KUKA KRL program: Work_2.src, Work_2.dat

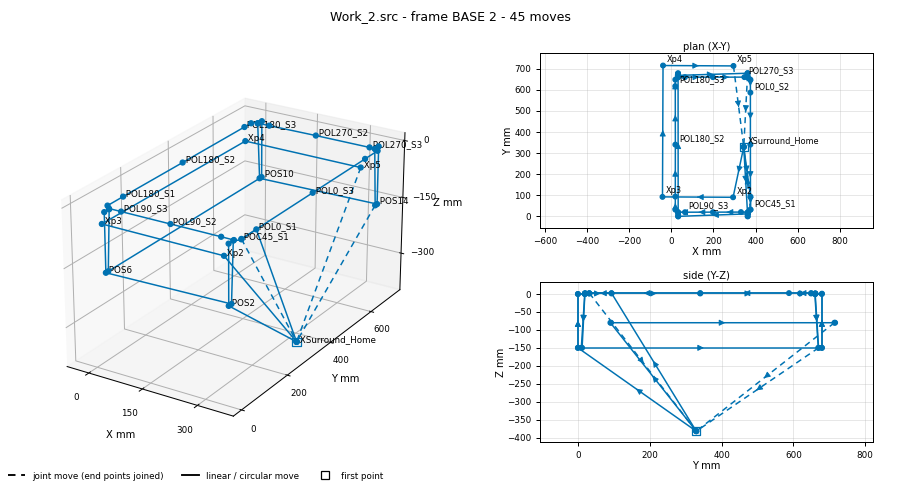
[picture p0: tool path of Work_2.src in frame BASE 2, 45 of 45 moves have a stored position in this frame; points joined in program order, loops and branches not executed]
--- Work_2.src ---
&ACCESS RVO1
&REL 406
&PARAM EDITMASK = *
&PARAM TEMPLATE = C:\KRC\Roboter\Template\vorgabe
&PARAM DISKPATH = KRC:\R1\KRL_HanGao\HG
DEF Work_2( )
;FOLD INI;%{PE}
  ;FOLD BASISTECH INI
    GLOBAL INTERRUPT DECL 3 WHEN $STOPMESS==TRUE DO IR_STOPM ( )
    INTERRUPT ON 3
    BAS (#INITMOV,0 )
  ;ENDFOLD (BASISTECH INI)
  ;FOLD USER INI
    ;Make your modifications here

  ;ENDFOLD (USER INI)
;ENDFOLD (INI)

;FOLD Vision.Vision_Ini ;%{PE}%MKUKATPUSER




EKRL_Vision_Int_Data("Xml_Ini_Data")


;ENDFOLD
;loop
;FOLD PTP Surround_Home Vel=20 % PDAT1 Tool[2]:Work_Tool Base[2]:B_2;%{PE}%R 8.3.48,%MKUKATPBASIS,%CMOVE,%VPTP,%P 1:PTP, 2:Surround_Home, 3:, 5:20, 7:PDAT1
$BWDSTART=FALSE
PDAT_ACT=PPDAT1
FDAT_ACT=FSurround_Home
BAS(#PTP_PARAMS,20)
PTP XSurround_Home
;ENDFOLD


;FOLD Vision.Camera_Offset Camera_NAME :P2, Area:45, Work:2;%{PE}%MKUKATPUSER

 HanGao_Camera_Offset(#Calibration ,1,2,XP2)





;ENDFOLD
;FOLD LIN p2 Vel=0.5 m/s CPDAT1 Tool[2]:Work_Tool Base[2]:Work_2 ;%{PE}
;FOLD Parameters ;%{h}
;Params IlfProvider=kukaroboter.basistech.inlineforms.movement.old; Kuka.IsGlobalPoint=False; Kuka.PointName=p2; Kuka.BlendingEnabled=False; Kuka.MoveDataName=CPDAT1; Kuka.VelocityPath=0.5; Kuka.CurrentCDSetIndex=0; Kuka.MovementParameterFieldEnabled=True; IlfCommand=LIN
;ENDFOLD
$BWDSTART = FALSE
LDAT_ACT = LCPDAT1
FDAT_ACT = Fp2
BAS(#CP_PARAMS, 0.5)
SET_CD_PARAMS (0)
LIN Xp2
;ENDFOLD
;FOLD Vision.Find_Model Work:2, Area:45;%{PE}%MKUKATPUSER



EKRL_Find_Model_Send("Xml_Vision_Model",2,1)



;ENDFOLD


;FOLD Vision.Camera_Offset Camera_NAME :P3, Area:135, Work:2;%{PE}%MKUKATPUSER

 HanGao_Camera_Offset(#Calibration ,2,2,XP3)





;ENDFOLD
;FOLD LIN p3 Vel=0.5 m/s CPDAT2 Tool[2]:Work_Tool Base[2]:Work_2 ;%{PE}
;FOLD Parameters ;%{h}
;Params IlfProvider=kukaroboter.basistech.inlineforms.movement.old; Kuka.IsGlobalPoint=False; Kuka.PointName=p3; Kuka.BlendingEnabled=False; Kuka.MoveDataName=CPDAT2; Kuka.VelocityPath=0.5; Kuka.CurrentCDSetIndex=0; Kuka.MovementParameterFieldEnabled=True; IlfCommand=LIN
;ENDFOLD
$BWDSTART = FALSE
LDAT_ACT = LCPDAT2
FDAT_ACT = Fp3
BAS(#CP_PARAMS, 0.5)
SET_CD_PARAMS (0)
LIN Xp3
;ENDFOLD
;FOLD Vision.Find_Model Work:2, Area:135;%{PE}%MKUKATPUSER



EKRL_Find_Model_Send("Xml_Vision_Model",2,2)



;ENDFOLD


;FOLD Vision.Camera_Offset Camera_NAME :P4, Area:225, Work:2;%{PE}%MKUKATPUSER

 HanGao_Camera_Offset(#Calibration ,3,2,XP4)





;ENDFOLD
;FOLD LIN p4 Vel=0.5 m/s CPDAT3 Tool[2]:Work_Tool Base[2]:Work_2 ;%{PE}
;FOLD Parameters ;%{h}
;Params IlfProvider=kukaroboter.basistech.inlineforms.movement.old; Kuka.IsGlobalPoint=False; Kuka.PointName=p4; Kuka.BlendingEnabled=False; Kuka.MoveDataName=CPDAT3; Kuka.VelocityPath=0.5; Kuka.CurrentCDSetIndex=0; Kuka.MovementParameterFieldEnabled=True; IlfCommand=LIN
;ENDFOLD
$BWDSTART = FALSE
LDAT_ACT = LCPDAT3
FDAT_ACT = Fp4
BAS(#CP_PARAMS, 0.5)
SET_CD_PARAMS (0)
LIN Xp4
;ENDFOLD
;FOLD Vision.Find_Model Work:2, Area:225;%{PE}%MKUKATPUSER



EKRL_Find_Model_Send("Xml_Vision_Model",2,3)



;ENDFOLD


;FOLD Vision.Camera_Offset Camera_NAME :P5, Area:315, Work:2;%{PE}%MKUKATPUSER

 HanGao_Camera_Offset(#Calibration ,4,2,XP5)





;ENDFOLD
;FOLD LIN p5 Vel=0.5 m/s CPDAT4 Tool[2]:Work_Tool Base[2]:Work_2 ;%{PE}
;FOLD Parameters ;%{h}
;Params IlfProvider=kukaroboter.basistech.inlineforms.movement.old; Kuka.IsGlobalPoint=False; Kuka.PointName=p5; Kuka.BlendingEnabled=False; Kuka.MoveDataName=CPDAT4; Kuka.VelocityPath=0.5; Kuka.CurrentCDSetIndex=0; Kuka.MovementParameterFieldEnabled=True; IlfCommand=LIN
;ENDFOLD
$BWDSTART = FALSE
LDAT_ACT = LCPDAT4
FDAT_ACT = Fp5
BAS(#CP_PARAMS, 0.5)
SET_CD_PARAMS (0)
LIN Xp5
;ENDFOLD
;FOLD Vision.Find_Model Work:2, Area:315;%{PE}%MKUKATPUSER



EKRL_Find_Model_Send("Xml_Vision_Model",2,4)



;ENDFOLD
;endloop
;halt
;FOLD PTP Surround_Home Vel=10 % PDAT4 Tool[2]:Work_Tool Base[2]:Work_2 ;%{PE}
;FOLD Parameters ;%{h}
;Params IlfProvider=kukaroboter.basistech.inlineforms.movement.old; Kuka.IsGlobalPoint=False; Kuka.PointName=Surround_Home; Kuka.BlendingEnabled=False; Kuka.MoveDataPtpName=PDAT4; Kuka.VelocityPtp=10; Kuka.CurrentCDSetIndex=0; Kuka.MovementParameterFieldEnabled=True; IlfCommand=PTP
;ENDFOLD
$BWDSTART = FALSE
PDAT_ACT = PPDAT4
FDAT_ACT = FSurround_Home
BAS(#PTP_PARAMS, 10.0)
SET_CD_PARAMS (0)
PTP XSurround_Home
;ENDFOLD
;FOLD Surround_LIN.S_LIN Point: L0_S1, Vel= 0.3 m/s, Point: 90 %, Area: LO, LDAT: L0_L1, OFFSET_NO: 1, Work: N_2 ;%{PE}
; LIN L0_S1POS: X=379.498230, Y=93.8288574, Z=1.00000, A=0.0, B=-20.0000, C=0.0
; LIN Offset POS:X=0.0, Y=0.0, Z=0.0
HanGao_Surr_Calculate( 90, #L0, #L_LIN_POS , POL0_S1, , , L0_Welding_Craft[2,1].Welding_Offset  , , 1, 2 )

HanGao_DAT_ACT(L0_Welding_Craft[2,1],LL0_L1)




FDAT_ACT=FL0_S1
LDAT_ACT=LL0_L1
BAS(#CP_PARAMS,L0_Welding_Craft[2,1].Welding_Speed )
LIN POL0_S1 C_DIS C_DIS
;ENDFOLD
;FOLD Laser_Function.LSON POW= 0 %, Sec= 0 S;%{PE}%MKUKATPUSER



  LSON(0/100,0)


;ENDFOLD
;FOLD Surround_LIN.S_C_LIN Point: C45_S1, Vel= 0.3 m/s, Area: C45, LDAT: C45_L1, Work: N_2 ;%{PE}
; CIR C45_S1POS: X=406.498535, Y=35.6358643, Z=0.0, A=0.0, B=20.0000, C=0.0
; CIR Offset POS:X=0.0, Y=0.0, Z=0.0
HanGao_Surr_Calculate(  , #C45, #C_LIN_POS , POC45_S1, , , C45_Welding_Craft[2,1].Welding_Offset , ,  , 2)

HanGao_DAT_ACT(C45_Welding_Craft[2,1],LC45_L1)




FDAT_ACT=FC45_S1
LDAT_ACT=LC45_L1
BAS(#CP_PARAMS, C45_Welding_Craft[2,1].Welding_Speed )
LIN POC45_S1 C_DIS C_DIS
;ENDFOLD
;FOLD Surround_CIR.S_C_CIR Point:PM3, PE3, Vel=.04m/s, Angle Area: C45, Work: N_2;%{PE}%MKUKATPUSER

; CIR MID POS:PM3 : X=0, Y=0, Z=0, A=0, B=0, C=0
; CIR END POS:PE3 : X=0, Y=0, Z=0, A=0, B=0, C=0
; CIR_MID_OFFSET  : X=0, Y=0, Z=0
; CIR_END_OFFSET  : X=0, Y=0, Z=0
HanGao_Surr_Calculate(  , #C45, #C_CIR_POS ,  , POPM3, POPE3 , C45_Welding_Craft[2,2].Welding_Offset  , C45_Welding_Craft[2, 3].Welding_Offset  ,  , 2)
TRIGGER WHEN PATH=0 DELAY=0 DO $ANOUT[1]=C45_Welding_Craft[2,3].Welding_Power/100

LPM3.VEL=C45_Welding_Craft[2,3].Welding_Speed
LPM3.ACC=C45_Welding_Craft[2,3].Welding_ACC
LPM3.APO_DIST=C45_Welding_Craft[2,3].Welding_CDIS

FDAT_ACT=FPE3
LDAT_ACT=LPM3
BAS(#CP_PARAMS,C45_Welding_Craft[2,3].Welding_Speed )
CIRC POPM3, POPE3 C_DIS C_DIS

;ENDFOLD
;FOLD Surround_LIN.S_LIN Point: L90_S1, Vel= 0.025 m/s, Point: 10 %, Area: L90, LDAT: L90_L1, OFFSET_NO: 1, Work: N_2 ;%{PE}
; LIN L90_S1POS: X=330.358398, Y=17.8462887, Z=1.00000, A=0.0, B=0.0, C=20.0000
; LIN Offset POS:X=0.0, Y=0.200000, Z=0.0
HanGao_Surr_Calculate( 10, #L90, #L_LIN_POS , POL90_S1, , , L90_Welding_Craft[2,1].Welding_Offset  , , 1, 2 )

HanGao_DAT_ACT(L90_Welding_Craft[2,1],LL90_L1)




FDAT_ACT=FL90_S1
LDAT_ACT=LL90_L1
BAS(#CP_PARAMS,L90_Welding_Craft[2,1].Welding_Speed )
LIN POL90_S1 C_DIS C_DIS
;ENDFOLD
;FOLD Surround_LIN.S_LIN Point: L90_S2, Vel= 0.025 m/s, Point: 50 %, Area: L90, LDAT: L90_L2, OFFSET_NO: 2, Work: N_2 ;%{PE}
; LIN L90_S2POS: X=0.0, Y=0.0, Z=0.0, A=0.0, B=0.0, C=0.0
; LIN Offset POS:X=0.0, Y=0.200000, Z=0.0
HanGao_Surr_Calculate( 50, #L90, #L_LIN_POS , POL90_S2, , , L90_Welding_Craft[2,2].Welding_Offset  , , 2, 2 )

HanGao_DAT_ACT(L90_Welding_Craft[2,2],LL90_L2)




FDAT_ACT=FL90_S2
LDAT_ACT=LL90_L2
BAS(#CP_PARAMS,L90_Welding_Craft[2,2].Welding_Speed )
LIN POL90_S2 C_DIS C_DIS
;ENDFOLD
;FOLD Surround_LIN.S_LIN Point: L90_S3, Vel= 0.025 m/s, Point: 90 %, Area: L90, LDAT: L90_L3, OFFSET_NO: 3, Work: N_2 ;%{PE}
; LIN L90_S3POS: X=0.0, Y=0.0, Z=0.0, A=0.0, B=0.0, C=0.0
; LIN Offset POS:X=0.0, Y=0.200000, Z=0.0
HanGao_Surr_Calculate( 90, #L90, #L_LIN_POS , POL90_S3, , , L90_Welding_Craft[2,3].Welding_Offset  , , 3, 2 )

HanGao_DAT_ACT(L90_Welding_Craft[2,3],LL90_L3)




FDAT_ACT=FL90_S3
LDAT_ACT=LL90_L3
BAS(#CP_PARAMS,L90_Welding_Craft[2,3].Welding_Speed )
LIN POL90_S3 C_DIS C_DIS
;ENDFOLD
;FOLD Surround_LIN.S_C_LIN Point: C135_S1, Vel= 0.2 m/s, Area: C135, LDAT: C135_L1, Work: N_2 ;%{PE}
; CIR C135_S1POS: X=0.0, Y=0.0, Z=0.0, A=0.0, B=0.0, C=0.0
; CIR Offset POS:X=-0.500000, Y=0.0, Z=0.0
HanGao_Surr_Calculate(  , #C135, #C_LIN_POS , POC135_S1, , , C135_Welding_Craft[2,1].Welding_Offset , ,  , 2)

HanGao_DAT_ACT(C135_Welding_Craft[2,1],LC135_L1)




FDAT_ACT=FC135_S1
LDAT_ACT=LC135_L1
BAS(#CP_PARAMS, C135_Welding_Craft[2,1].Welding_Speed )
LIN POC135_S1 C_DIS C_DIS
;ENDFOLD
;FOLD Surround_CIR.S_C_CIR Point: PM4, PE4, Vel= 0.012 m/s, Angle Area: C135, Work: N_2 ;%{PE}
; CIR MID POS:PM4 : X=22.6620, Y=25.2540, Z=1.00000, A=0.0, B=0.0, C=0.0
; CIR END POS:PE4 : X=20.6667957, Y=33.6577797, Z=0.0, A=0.0, B=-20.0000, C=0.0
; CIR_MID_OFFSET  : X=0.0, Y=0.0, Z=0.0
; CIR_END_OFFSET  : X=0.500000, Y=0.0, Z=-1.00000
HanGao_Surr_Calculate(  , #C135, #C_CIR_POS ,  , POPM4, POPE4 , C135_Welding_Craft[2,2].Welding_Offset  , C135_Welding_Craft[2, 3].Welding_Offset  ,  , 2)

HanGao_DAT_ACT(C135_Welding_Craft[2,3],LPM4)




FDAT_ACT=FPE4
LDAT_ACT=LPM4
BAS(#CP_PARAMS,C135_Welding_Craft[2,3].Welding_Speed )
CIRC POPM4, POPE4 C_DIS C_DIS
;ENDFOLD
;FOLD Surround_LIN.S_LIN Point: L180_S1, Vel= 0.025 m/s, Point: 10 %, Area: L180, LDAT: L180_L1, OFFSET_NO: 1, Work: N_2 ;%{PE}
; LIN L180_S1POS: X=20.5413361, Y=95.3976288, Z=0.0, A=0.0, B=-20.0000, C=0.0
; LIN Offset POS:X=0.0, Y=0.0, Z=-1.00000
HanGao_Surr_Calculate( 10, #L180, #L_LIN_POS , POL180_S1, , , L180_Welding_Craft[2,1].Welding_Offset  , , 1, 2 )

HanGao_DAT_ACT(L180_Welding_Craft[2,1],LL180_L1)




FDAT_ACT=FL180_S1
LDAT_ACT=LL180_L1
BAS(#CP_PARAMS,L180_Welding_Craft[2,1].Welding_Speed )
LIN POL180_S1 C_DIS C_DIS
;ENDFOLD
;FOLD Surround_LIN.S_LIN Point: L180_S2, Vel= 0.03 m/s, Point: 50 %, Area: L180, LDAT: L180_L2, OFFSET_NO: 2, Work: N_2 ;%{PE}
; LIN L180_S2POS: X=22.3395, Y=342.357025, Z=0.0, A=0.0, B=-20.0000, C=0.0
; LIN Offset POS:X=0.300000, Y=0.0, Z=-1.00000
HanGao_Surr_Calculate( 50, #L180, #L_LIN_POS , POL180_S2, , , L180_Welding_Craft[2,2].Welding_Offset  , , 2, 2 )

HanGao_DAT_ACT(L180_Welding_Craft[2,2],LL180_L2)




FDAT_ACT=FL180_S2
LDAT_ACT=LL180_L2
BAS(#CP_PARAMS,L180_Welding_Craft[2,2].Welding_Speed )
LIN POL180_S2 C_DIS C_DIS
;ENDFOLD
;FOLD Surround_LIN.S_LIN Point: L180_S3, Vel= 0.03 m/s, Point: 95 %, Area: L180, LDAT: L180_L3, OFFSET_NO: 3, Work: N_2 ;%{PE}
; LIN L180_S3POS: X=24.0249329, Y=620.186340, Z=0.0, A=0.0, B=-20.0000, C=0.0
; LIN Offset POS:X=0.300000, Y=0.0, Z=-1.00000
HanGao_Surr_Calculate( 95, #L180, #L_LIN_POS , POL180_S3, , , L180_Welding_Craft[2,3].Welding_Offset  , , 3, 2 )

HanGao_DAT_ACT(L180_Welding_Craft[2,3],LL180_L3)




FDAT_ACT=FL180_S3
LDAT_ACT=LL180_L3
BAS(#CP_PARAMS,L180_Welding_Craft[2,3].Welding_Speed )
LIN POL180_S3 C_DIS C_DIS
;ENDFOLD
;FOLD Surround_LIN.S_C_LIN Point: C225_S1, Vel= 0.2 m/s, Area: C225, LDAT: C225_L1, Work: N_2 ;%{PE}
; CIR C225_S1POS: X=24.2122040, Y=651.056274, Z=0.0, A=0.0, B=-20.0000, C=0.0
; CIR Offset POS:X=-0.500000, Y=0.0, Z=0.0
HanGao_Surr_Calculate(  , #C225, #C_LIN_POS , POC225_S1, , , C225_Welding_Craft[2,1].Welding_Offset , ,  , 2)

HanGao_DAT_ACT(C225_Welding_Craft[2,1],LC225_L1)




FDAT_ACT=FC225_S1
LDAT_ACT=LC225_L1
BAS(#CP_PARAMS, C225_Welding_Craft[2,1].Welding_Speed )
LIN POC225_S1 C_DIS C_DIS
;ENDFOLD
;FOLD Surround_CIR.S_C_CIR Point: PM5, PE5, Vel= 0.012 m/s, Angle Area: C225, Work: N_2 ;%{PE}
; CIR MID POS:PM5 : X=28.3490, Y=660.056, Z=1.00000, A=0.0, B=0.0, C=0.0
; CIR END POS:PE5 : X=35.9848671, Y=663.799744, Z=1.00000, A=0.0, B=0.0, C=-20.0000
; CIR_MID_OFFSET  : X=0.0, Y=0.500000, Z=0.0
; CIR_END_OFFSET  : X=0.0, Y=0.800000, Z=0.0
HanGao_Surr_Calculate(  , #C225, #C_CIR_POS ,  , POPM5, POPE5 , C225_Welding_Craft[2,2].Welding_Offset  , C225_Welding_Craft[2, 3].Welding_Offset  ,  , 2)

HanGao_DAT_ACT(C225_Welding_Craft[2,3],LPM5)




FDAT_ACT=FPE5
LDAT_ACT=LPM5
BAS(#CP_PARAMS,C225_Welding_Craft[2,3].Welding_Speed )
CIRC POPM5, POPE5 C_DIS C_DIS
;ENDFOLD
;FOLD Surround_LIN.S_LIN Point: L270_S1, Vel= 0.025 m/s, Point: 10 %, Area: L270, LDAT: l270_L1, OFFSET_NO: 1, Work: N_2 ;%{PE}
; LIN L270_S1POS: X=69.2440872, Y=662.843689, Z=1.00000, A=0.0, B=0.0, C=-20.0000
; LIN Offset POS:X=0.0, Y=0.0, Z=0.0
HanGao_Surr_Calculate( 10, #L270, #L_LIN_POS , POL270_S1, , , L270_Welding_Craft[2,1].Welding_Offset  , , 1, 2 )

HanGao_DAT_ACT(L270_Welding_Craft[2,1],Ll270_L1)




FDAT_ACT=FL270_S1
LDAT_ACT=Ll270_L1
BAS(#CP_PARAMS,L270_Welding_Craft[2,1].Welding_Speed )
LIN POL270_S1 C_DIS C_DIS
;ENDFOLD
;FOLD Surround_LIN.S_LIN Point: L270_S2, Vel= 0.03 m/s, Point: 50 %, Area: L270, LDAT: L270_L2, OFFSET_NO: 2, Work: N_2 ;%{PE}
; LIN L270_S2POS: X=202.280975, Y=661.419495, Z=1.00000, A=0.0, B=0.0, C=-20.0000
; LIN Offset POS:X=0.0, Y=-0.800000, Z=0.0
HanGao_Surr_Calculate( 50, #L270, #L_LIN_POS , POL270_S2, , , L270_Welding_Craft[2,2].Welding_Offset  , , 2, 2 )

HanGao_DAT_ACT(L270_Welding_Craft[2,2],LL270_L2)




FDAT_ACT=FL270_S2
LDAT_ACT=LL270_L2
BAS(#CP_PARAMS,L270_Welding_Craft[2,2].Welding_Speed )
LIN POL270_S2 C_DIS C_DIS
;ENDFOLD
;FOLD Surround_LIN.S_LIN Point: L270_S3, Vel= 0.03 m/s, Point: 95 %, Area: L270, LDAT: L270_L3, OFFSET_NO: 3, Work: N_2 ;%{PE}
; LIN L270_S3POS: X=351.947479, Y=660.717285, Z=1.00000, A=0.0, B=0.0, C=-20.0000
; LIN Offset POS:X=0.0, Y=-0.800000, Z=0.0
HanGao_Surr_Calculate( 95, #L270, #L_LIN_POS , POL270_S3, , , L270_Welding_Craft[2,3].Welding_Offset  , , 3, 2 )

HanGao_DAT_ACT(L270_Welding_Craft[2,3],LL270_L3)




FDAT_ACT=FL270_S3
LDAT_ACT=LL270_L3
BAS(#CP_PARAMS,L270_Welding_Craft[2,3].Welding_Speed )
LIN POL270_S3 C_DIS C_DIS
;ENDFOLD
;FOLD Surround_LIN.S_C_LIN Point: C315_S1, Vel= 0.2 m/s, Area: C315, LDAT: C315_L1, Work: N_2 ;%{PE}
; CIR C315_S1POS: X=368.577087, Y=660.939270, Z=1.00000, A=0.0, B=0.0, C=-20.0000
; CIR Offset POS:X=-0.500000, Y=0.0, Z=0.0
HanGao_Surr_Calculate(  , #C315, #C_LIN_POS , POC315_S1, , , C315_Welding_Craft[2,1].Welding_Offset , ,  , 2)

HanGao_DAT_ACT(C315_Welding_Craft[2,1],LC315_L1)




FDAT_ACT=FC315_S1
LDAT_ACT=LC315_L1
BAS(#CP_PARAMS, C315_Welding_Craft[2,1].Welding_Speed )
LIN POC315_S1 C_DIS C_DIS
;ENDFOLD
;FOLD Surround_CIR.S_C_CIR Point: PM7, PE7, Vel= 0.012 m/s, Angle Area: C315, Work: N_2 ;%{PE}
; CIR MID POS:PM7 : X=377.618, Y=656.195, Z=1.00000, A=0.0, B=0.0, C=0.0
; CIR END POS:PE7 : X=380.001862, Y=649.383240, Z=1.00000, A=0.0, B=20.0000, C=0.0
; CIR_MID_OFFSET  : X=0.0, Y=-0.500000, Z=0.0
; CIR_END_OFFSET  : X=-0.500000, Y=0.0, Z=0.0
HanGao_Surr_Calculate(  , #C315, #C_CIR_POS ,  , POPM7, POPE7 , C315_Welding_Craft[2,2].Welding_Offset  , C315_Welding_Craft[2, 3].Welding_Offset  ,  , 2)

HanGao_DAT_ACT(C315_Welding_Craft[2,3],LPM7)




FDAT_ACT=FPE7
LDAT_ACT=LPM7
BAS(#CP_PARAMS,C315_Welding_Craft[2,3].Welding_Speed )
CIRC POPM7, POPE7 C_DIS C_DIS
;ENDFOLD
;FOLD Surround_LIN.S_LIN Point: L0_S2, Vel= 0.03 m/s, Point: 10 %, Area: LO, LDAT: L0_L2, OFFSET_NO: 2, Work: N_2 ;%{PE}
; LIN L0_S2POS: X=379.614777, Y=587.556091, Z=1.00000, A=0.0, B=20.0000, C=0.0
; LIN Offset POS:X=-0.500000, Y=0.0, Z=0.0
HanGao_Surr_Calculate( 10, #L0, #L_LIN_POS , POL0_S2, , , L0_Welding_Craft[2,2].Welding_Offset  , , 2, 2 )

HanGao_DAT_ACT(L0_Welding_Craft[2,2],LL0_L2)




FDAT_ACT=FL0_S2
LDAT_ACT=LL0_L2
BAS(#CP_PARAMS,L0_Welding_Craft[2,2].Welding_Speed )
LIN POL0_S2 C_DIS C_DIS
;ENDFOLD
;FOLD Surround_LIN.S_LIN Point: L0_S3, Vel= 0.03 m/s, Point: 50 %, Area: LO, LDAT: L0_L3, OFFSET_NO: 3, Work: N_2 ;%{PE}
; LIN L0_S3POS: X=378.066498, Y=340.247498, Z=1.00000, A=0.0, B=20.0000, C=0.0
; LIN Offset POS:X=-0.500000, Y=0.0, Z=0.0
HanGao_Surr_Calculate( 50, #L0, #L_LIN_POS , POL0_S3, , , L0_Welding_Craft[2,3].Welding_Offset  , , 3, 2 )

HanGao_DAT_ACT(L0_Welding_Craft[2,3],LL0_L3)




FDAT_ACT=FL0_S3
LDAT_ACT=LL0_L3
BAS(#CP_PARAMS,L0_Welding_Craft[2,3].Welding_Speed )
LIN POL0_S3 C_DIS C_DIS
;ENDFOLD
;FOLD Surround_LIN.S_LIN Point: L0_S4, Vel= 0.04 m/s, Point: 100 %, Area: LO, LDAT: L0_L4, OFFSET_NO: 4, Work: N_2 ;%{PE}
; LIN L0_S4POS: X=375.599823, Y=62.1482544, Z=2.50000, A=0.0, B=20.0000, C=0.0
; LIN Offset POS:X=-0.200000, Y=0.0, Z=1.00000
HanGao_Surr_Calculate( 100, #L0, #L_LIN_POS , POL0_S4, , , L0_Welding_Craft[2,4].Welding_Offset  , , 4, 2 )

HanGao_DAT_ACT(L0_Welding_Craft[2,4],LL0_L4)




FDAT_ACT=FL0_S4
LDAT_ACT=LL0_L4
BAS(#CP_PARAMS,L0_Welding_Craft[2,4].Welding_Speed )
LIN POL0_S4 C_DIS C_DIS
;ENDFOLD
;FOLD Laser_Function.LSOFF ;%{PE}%MKUKATPUSER


   LSOFF()


;ENDFOLD


;FOLD PTP Surround_Home Vel=10 % PDAT2 Tool[2]:Work_Tool Base[2]:B_2;%{PE}%R 8.3.48,%MKUKATPBASIS,%CMOVE,%VPTP,%P 1:PTP, 2:Surround_Home, 3:, 5:10, 7:PDAT2
$BWDSTART=FALSE
PDAT_ACT=PPDAT2
FDAT_ACT=FSurround_Home
BAS(#PTP_PARAMS,10)
PTP XSurround_Home
;ENDFOLD
if (false) THEN
;halt
;return
;FOLD Short_Craft.S_LIN Point: S2, Vel= 0.5 m/s, Area: N45, Short_Pos: Safety, Point: 50 %, LDAT: L2, Work: N_2 ;%{PE}
; LIN S2POS: X=363.220, Y=-0.316000, Z=-150.000, A=0.0, B=0.0, C=0.0
; LIN Offset POS:X=0.0, Y=0.0, Z=0.0
HanGao_Surr_Calculate( 50, #N45, #L_LIN_POS , POS2, , , N45_Short_Craft[2,1].Welding_Offset  , , 1, 2, N2_Sink_Data.Sink_Type)

HanGao_DAT_ACT(N45_Short_Craft[2,1],LL2)




FDAT_ACT=FS2
LDAT_ACT=LL2
BAS(#CP_PARAMS,N45_Short_Craft[2,1].Welding_Speed )
LIN POS2 C_DIS C_DIS
;ENDFOLD
;FOLD Short_Craft.S_LIN Point: S3, Vel= 0.5 m/s, Area: N45, Short_Pos: Start, Point: 50 %, LDAT: L3, Work: N_2 ;%{PE}
; LIN S3POS: X=363.220, Y=-0.316000, Z=0.0, A=0.0, B=0.0, C=0.0
; LIN Offset POS:X=0.0, Y=0.0, Z=0.0
HanGao_Surr_Calculate( 50, #N45, #L_LIN_POS , POS3, , , N45_Short_Craft[2,2].Welding_Offset  , , 2, 2, N2_Sink_Data.Sink_Type)

HanGao_DAT_ACT(N45_Short_Craft[2,2],LL3)




FDAT_ACT=FS3
LDAT_ACT=LL3
BAS(#CP_PARAMS,N45_Short_Craft[2,2].Welding_Speed )
LIN POS3 C_DIS C_DIS
;ENDFOLD
;FOLD Laser_Function.LSON POW= .5 %, Sec= 0 S;%{PE}%MKUKATPUSER



  LSON(.5/100,0)


;ENDFOLD
;FOLD Short_Craft.S_LIN Point: S4, Vel= 0.01 m/s, Area: N45, Short_Pos: End, Point: 50 %, LDAT: L4, Work: N_2 ;%{PE}
; LIN S4POS: X=363.395, Y=19.3140, Z=0.0, A=0.0, B=0.0, C=0.0
; LIN Offset POS:X=0.0, Y=0.0, Z=0.0
HanGao_Surr_Calculate( 50, #N45, #L_LIN_POS , POS4, , , N45_Short_Craft[2,3].Welding_Offset  , , 3, 2, N2_Sink_Data.Sink_Type)

HanGao_DAT_ACT(N45_Short_Craft[2,3],LL4)




FDAT_ACT=FS4
LDAT_ACT=LL4
BAS(#CP_PARAMS,N45_Short_Craft[2,3].Welding_Speed )
LIN POS4 C_DIS C_DIS
;ENDFOLD
;FOLD Short_Craft.S_LIN Point: S5, Vel= 0.5 m/s, Area: N45, Short_Pos: BackWelding, Point: 10 %, LDAT: L5, Work: N_2 ;%{PE}
; LIN S5POS: X=363.323059, Y=11.2466183, Z=-150.000, A=0.0, B=0.0, C=0.0
; LIN Offset POS:X=0.0, Y=0.0, Z=0.0
HanGao_Surr_Calculate( 10, #N45, #L_LIN_POS , POS5, , , N45_Short_Craft[2,4].Welding_Offset  , , 4, 2, N2_Sink_Data.Sink_Type)

HanGao_DAT_ACT(N45_Short_Craft[2,4],LL5)




FDAT_ACT=FS5
LDAT_ACT=LL5
BAS(#CP_PARAMS,N45_Short_Craft[2,4].Welding_Speed )
LIN POS5 C_DIS C_DIS
;ENDFOLD
;FOLD Laser_Function.LSOFF ;%{PE}%MKUKATPUSER


   LSOFF()


;ENDFOLD


;FOLD Short_Craft.S_LIN Point: S6, Vel= 0.5 m/s, Area: N135, Short_Pos: Safety, Point: 50 %, LDAT: L6, Work: N_2 ;%{PE}
; LIN S6POS: X=32.5260, Y=-0.971000, Z=-150.000, A=0.0, B=0.0, C=0.0
; LIN Offset POS:X=0.0, Y=0.0, Z=0.0
HanGao_Surr_Calculate( 50, #N135, #L_LIN_POS , POS6, , , N135_Short_Craft[2,1].Welding_Offset  , , 1, 2, N2_Sink_Data.Sink_Type)

HanGao_DAT_ACT(N135_Short_Craft[2,1],LL6)




FDAT_ACT=FS6
LDAT_ACT=LL6
BAS(#CP_PARAMS,N135_Short_Craft[2,1].Welding_Speed )
LIN POS6 C_DIS C_DIS
;ENDFOLD
;FOLD Short_Craft.S_LIN Point: S7, Vel= 0.5 m/s, Area: N135, Short_Pos: Start, Point: 50 %, LDAT: L7, Work: N_2 ;%{PE}
; LIN S7POS: X=32.5260, Y=-0.971000, Z=0.0, A=0.0, B=0.0, C=0.0
; LIN Offset POS:X=0.0, Y=0.0, Z=0.0
HanGao_Surr_Calculate( 50, #N135, #L_LIN_POS , POS7, , , N135_Short_Craft[2,2].Welding_Offset  , , 2, 2, N2_Sink_Data.Sink_Type)

HanGao_DAT_ACT(N135_Short_Craft[2,2],LL7)




FDAT_ACT=FS7
LDAT_ACT=LL7
BAS(#CP_PARAMS,N135_Short_Craft[2,2].Welding_Speed )
LIN POS7 C_DIS C_DIS
;ENDFOLD
;FOLD Laser_Function.LSON POW= 60 %, Sec= 0 S;%{PE}%MKUKATPUSER



  LSON(60/100,0)


;ENDFOLD
;FOLD Short_Craft.S_LIN Point: S8, Vel= 0.01 m/s, Area: N135, Short_Pos: End, Point: 50 %, LDAT: L8, Work: N_2 ;%{PE}
; LIN S8POS: X=32.3940, Y=18.1940, Z=0.0, A=0.0, B=0.0, C=0.0
; LIN Offset POS:X=0.0, Y=0.0, Z=0.0
HanGao_Surr_Calculate( 50, #N135, #L_LIN_POS , POS8, , , N135_Short_Craft[2,3].Welding_Offset  , , 3, 2, N2_Sink_Data.Sink_Type)

HanGao_DAT_ACT(N135_Short_Craft[2,3],LL8)




FDAT_ACT=FS8
LDAT_ACT=LL8
BAS(#CP_PARAMS,N135_Short_Craft[2,3].Welding_Speed )
LIN POS8 C_DIS C_DIS
;ENDFOLD
;FOLD Short_Craft.S_LIN Point: S9, Vel= 0.5 m/s, Area: N135, Short_Pos: BackWelding, Point: 50 %, LDAT: L9, Work: N_2 ;%{PE}
; LIN S9POS: X=32.4600, Y=8.61150074, Z=-150.000, A=0.0, B=0.0, C=0.0
; LIN Offset POS:X=0.0, Y=0.0, Z=0.0
HanGao_Surr_Calculate( 50, #N135, #L_LIN_POS , POS9, , , N135_Short_Craft[2,4].Welding_Offset  , , 4, 2, N2_Sink_Data.Sink_Type)

HanGao_DAT_ACT(N135_Short_Craft[2,4],LL9)




FDAT_ACT=FS9
LDAT_ACT=LL9
BAS(#CP_PARAMS,N135_Short_Craft[2,4].Welding_Speed )
LIN POS9 C_DIS C_DIS
;ENDFOLD
;FOLD Laser_Function.LSOFF ;%{PE}%MKUKATPUSER


   LSOFF()


;ENDFOLD


;FOLD Short_Craft.S_LIN Point: S10, Vel= 0.5 m/s, Area: N225, Short_Pos: Safety, Point: 50 %, LDAT: L10, Work: N_2 ;%{PE}
; LIN S10POS: X=31.6330, Y=679.439, Z=-150.000, A=0.0, B=0.0, C=0.0
; LIN Offset POS:X=0.0, Y=0.0, Z=0.0
HanGao_Surr_Calculate( 50, #N225, #L_LIN_POS , POS10, , , N225_Short_Craft[2,1].Welding_Offset  , , 1, 2, N2_Sink_Data.Sink_Type)

HanGao_DAT_ACT(N225_Short_Craft[2,1],LL10)




FDAT_ACT=FS10
LDAT_ACT=LL10
BAS(#CP_PARAMS,N225_Short_Craft[2,1].Welding_Speed )
LIN POS10 C_DIS C_DIS
;ENDFOLD
;FOLD Short_Craft.S_LIN Point: S11, Vel= 0.5 m/s, Area: N225, Short_Pos: Start, Point: 50 %, LDAT: L11, Work: N_2 ;%{PE}
; LIN S11POS: X=31.6330, Y=679.439, Z=0.0, A=0.0, B=0.0, C=0.0
; LIN Offset POS:X=0.0, Y=0.0, Z=0.0
HanGao_Surr_Calculate( 50, #N225, #L_LIN_POS , POS11, , , N225_Short_Craft[2,2].Welding_Offset  , , 2, 2, N2_Sink_Data.Sink_Type)

HanGao_DAT_ACT(N225_Short_Craft[2,2],LL11)




FDAT_ACT=FS11
LDAT_ACT=LL11
BAS(#CP_PARAMS,N225_Short_Craft[2,2].Welding_Speed )
LIN POS11 C_DIS C_DIS
;ENDFOLD
;FOLD Laser_Function.LSON POW= 60 %, Sec= 0 S;%{PE}%MKUKATPUSER



  LSON(60/100,0)


;ENDFOLD
;FOLD Short_Craft.S_LIN Point: S12, Vel= 0.01 m/s, Area: N225, Short_Pos: End, Point: 50 %, LDAT: L12, Work: N_2 ;%{PE}
; LIN S12POS: X=31.8670, Y=660.025, Z=0.0, A=0.0, B=0.0, C=0.0
; LIN Offset POS:X=0.0, Y=0.0, Z=0.0
HanGao_Surr_Calculate( 50, #N225, #L_LIN_POS , POS12, , , N225_Short_Craft[2,3].Welding_Offset  , , 3, 2, N2_Sink_Data.Sink_Type)

HanGao_DAT_ACT(N225_Short_Craft[2,3],LL12)




FDAT_ACT=FS12
LDAT_ACT=LL12
BAS(#CP_PARAMS,N225_Short_Craft[2,3].Welding_Speed )
LIN POS12 C_DIS C_DIS
;ENDFOLD
;FOLD Short_Craft.S_LIN Point: S13, Vel= 0.5 m/s, Area: N225, Short_Pos: BackWelding, Point: 50 %, LDAT: L13, Work: N_2 ;%{PE}
; LIN S13POS: X=31.7500, Y=669.732056, Z=-150.000, A=0.0, B=0.0, C=0.0
; LIN Offset POS:X=0.0, Y=0.0, Z=0.0
HanGao_Surr_Calculate( 50, #N225, #L_LIN_POS , POS13, , , N225_Short_Craft[2,4].Welding_Offset  , , 4, 2, N2_Sink_Data.Sink_Type)

HanGao_DAT_ACT(N225_Short_Craft[2,4],LL13)




FDAT_ACT=FS13
LDAT_ACT=LL13
BAS(#CP_PARAMS,N225_Short_Craft[2,4].Welding_Speed )
LIN POS13 C_DIS C_DIS
;ENDFOLD
;FOLD Laser_Function.LSOFF ;%{PE}%MKUKATPUSER


   LSOFF()


;ENDFOLD


;FOLD Short_Craft.S_LIN Point: S14, Vel= 0.5 m/s, Area: N315, Short_Pos: Safety, Point: 50 %, LDAT: L14, Work: N_2 ;%{PE}
; LIN S14POS: X=362.986, Y=679.910, Z=-150.000, A=0.0, B=0.0, C=0.0
; LIN Offset POS:X=0.0, Y=0.0, Z=0.0
HanGao_Surr_Calculate( 50, #N315, #L_LIN_POS , POS14, , , N315_Short_Craft[2,1].Welding_Offset  , , 1, 2, N2_Sink_Data.Sink_Type)

HanGao_DAT_ACT(N315_Short_Craft[2,1],LL14)




FDAT_ACT=FS14
LDAT_ACT=LL14
BAS(#CP_PARAMS,N315_Short_Craft[2,1].Welding_Speed )
LIN POS14 C_DIS C_DIS
;ENDFOLD
;FOLD Short_Craft.S_LIN Point: S15, Vel= 0.5 m/s, Area: N315, Short_Pos: Start, Point: 50 %, LDAT: L15, Work: N_2 ;%{PE}
; LIN S15POS: X=362.986, Y=679.910, Z=1.00000, A=0.0, B=0.0, C=0.0
; LIN Offset POS:X=0.0, Y=0.0, Z=1.00000
HanGao_Surr_Calculate( 50, #N315, #L_LIN_POS , POS15, , , N315_Short_Craft[2,2].Welding_Offset  , , 2, 2, N2_Sink_Data.Sink_Type)

HanGao_DAT_ACT(N315_Short_Craft[2,2],LL15)




FDAT_ACT=FS15
LDAT_ACT=LL15
BAS(#CP_PARAMS,N315_Short_Craft[2,2].Welding_Speed )
LIN POS15 C_DIS C_DIS
;ENDFOLD
;FOLD Laser_Function.LSON POW= 60 %, Sec= 0 S;%{PE}%MKUKATPUSER



  LSON(60/100,0)


;ENDFOLD
;FOLD Short_Craft.S_LIN Point: S16, Vel= 0.01 m/s, Area: N315, Short_Pos: End, Point: 50 %, LDAT: L16, Work: N_2 ;%{PE}
; LIN S16POS: X=363.044, Y=660.468, Z=1.00000, A=0.0, B=0.0, C=0.0
; LIN Offset POS:X=0.0, Y=0.0, Z=1.00000
HanGao_Surr_Calculate( 50, #N315, #L_LIN_POS , POS16, , , N315_Short_Craft[2,3].Welding_Offset  , , 3, 2, N2_Sink_Data.Sink_Type)

HanGao_DAT_ACT(N315_Short_Craft[2,3],LL16)




FDAT_ACT=FS16
LDAT_ACT=LL16
BAS(#CP_PARAMS,N315_Short_Craft[2,3].Welding_Speed )
LIN POS16 C_DIS C_DIS
;ENDFOLD
;FOLD Short_Craft.S_LIN Point: S17, Vel= 0.5 m/s, Area: N315, Short_Pos: BackWelding, Point: 50 %, LDAT: L17, Work: N_2 ;%{PE}
; LIN S17POS: X=363.015, Y=670.188965, Z=-150.000, A=0.0, B=0.0, C=0.0
; LIN Offset POS:X=0.0, Y=0.0, Z=0.0
HanGao_Surr_Calculate( 50, #N315, #L_LIN_POS , POS17, , , N315_Short_Craft[2,4].Welding_Offset  , , 4, 2, N2_Sink_Data.Sink_Type)

HanGao_DAT_ACT(N315_Short_Craft[2,4],LL17)




FDAT_ACT=FS17
LDAT_ACT=LL17
BAS(#CP_PARAMS,N315_Short_Craft[2,4].Welding_Speed )
LIN POS17 C_DIS C_DIS
;ENDFOLD
;FOLD Laser_Function.LSOFF ;%{PE}%MKUKATPUSER


   LSOFF()


;ENDFOLD
endif

;FOLD PTP Surround_Home CONT Vel=30 % PDAT3 Tool[2]:Work_Tool Base[2]:B_2;%{PE}%R 8.3.48,%MKUKATPBASIS,%CMOVE,%VPTP,%P 1:PTP, 2:Surround_Home, 3:C_DIS, 5:30, 7:PDAT3
$BWDSTART=FALSE
PDAT_ACT=PPDAT3
FDAT_ACT=FSurround_Home
BAS(#PTP_PARAMS,30)
PTP XSurround_Home C_DIS
;ENDFOLD
END

--- Work_2.dat ---
&ACCESS RVO1
&REL 406
&PARAM EDITMASK = *
&PARAM TEMPLATE = C:\KRC\Roboter\Template\vorgabe
&PARAM DISKPATH = KRC:\R1\KRL_HanGao\HG
DEFDAT  WORK_2
;FOLD EXTERNAL DECLARATIONS;%{PE}%MKUKATPBASIS,%CEXT,%VCOMMON,%P
;FOLD BASISTECH EXT;%{PE}%MKUKATPBASIS,%CEXT,%VEXT,%P
EXT  BAS (BAS_COMMAND  :IN,REAL  :IN )
DECL INT SUCCESS
;ENDFOLD (BASISTECH EXT)
;FOLD USER EXT;%{E}%MKUKATPUSER,%CEXT,%VEXT,%P
;Make your modifications here

;ENDFOLD (USER EXT)
;ENDFOLD (EXTERNAL DECLARATIONS)
DECL BASIS_SUGG_T LAST_BASIS={POINT1[] "P0                      ",POINT2[] "P0                      ",CP_PARAMS[] "CPDAT0                  ",PTP_PARAMS[] "PDAT0                   ",CONT[] "                        ",CP_VEL[] "2.0                     ",PTP_VEL[] "100                     ",SYNC_PARAMS[] "SYNCDAT                 ",SPL_NAME[] "S0                      ",A_PARAMS[] "ADAT0                   "}
DECL E6POS XSURROUND_HOME={X 343.780548,Y 329.155823,Z -382.275,A 0.441927075,B -0.0416149125,C -0.0704164580,S 2,T 10,E1 0.0,E2 0.0,E3 0.0,E4 0.0,E5 0.0,E6 0.0}
DECL FDAT FSurround_Home={TOOL_NO 2,BASE_NO 2,IPO_FRAME #BASE,POINT2[] " "}
DECL PDAT PPDAT1={VEL 100.000,ACC 20.0000,APO_DIST 100.000,GEAR_JERK 50.0000,EXAX_IGN 0}
DECL PDAT PPDAT2={VEL 100.000,ACC 20.0000,APO_DIST 100.000,GEAR_JERK 50.0000,EXAX_IGN 0}
DECL E6POS POS2={X 362.596,Y -0.482000,Z -150.000,A 0.0,B 0.0,C 0.0}
DECL FDAT FS2={TOOL_NO 2,BASE_NO 2,IPO_FRAME #BASE,POINT2[] " ",TQ_STATE FALSE}
DECL LDAT LL2={VEL 0.500000,ACC 100.000,APO_DIST 0.0,APO_FAC 50.0000,AXIS_VEL 100.000,AXIS_ACC 100.000,ORI_TYP #VAR,CIRC_TYP #BASE,JERK_FAC 50.0000,GEAR_JERK 50.0000,EXAX_IGN 0}
DECL E6POS POS3={X 362.596,Y -0.482000,Z 0.0,A 0.0,B 0.0,C 0.0}
DECL FDAT FS3={TOOL_NO 2,BASE_NO 2,IPO_FRAME #BASE,POINT2[] " ",TQ_STATE FALSE}
DECL LDAT LL3={VEL 0.500000,ACC 100.000,APO_DIST 0.0,APO_FAC 50.0000,AXIS_VEL 100.000,AXIS_ACC 100.000,ORI_TYP #VAR,CIRC_TYP #BASE,JERK_FAC 50.0000,GEAR_JERK 50.0000,EXAX_IGN 0}
DECL E6POS POS4={X 362.546,Y 18.7470,Z 0.0,A 0.0,B 0.0,C 0.0}
DECL FDAT FS4={TOOL_NO 2,BASE_NO 2,IPO_FRAME #BASE,POINT2[] " ",TQ_STATE FALSE}
DECL LDAT LL4={VEL 0.01000000,ACC 100.000,APO_DIST 0.0,APO_FAC 50.0000,AXIS_VEL 100.000,AXIS_ACC 100.000,ORI_TYP #VAR,CIRC_TYP #BASE,JERK_FAC 50.0000,GEAR_JERK 50.0000,EXAX_IGN 0}
DECL E6POS POS5={X 362.566040,Y 11.0408678,Z -150.000,A 0.0,B 0.0,C 0.0}
DECL FDAT FS5={TOOL_NO 2,BASE_NO 2,IPO_FRAME #BASE,POINT2[] " ",TQ_STATE FALSE}
DECL LDAT LL5={VEL 0.500000,ACC 100.000,APO_DIST 0.0,APO_FAC 50.0000,AXIS_VEL 100.000,AXIS_ACC 100.000,ORI_TYP #VAR,CIRC_TYP #BASE,JERK_FAC 50.0000,GEAR_JERK 50.0000,EXAX_IGN 0}
DECL E6POS POPM3={X 372.487,Y 23.7200,Z 1.50000,A 0.0,B 0.0,C 0.0}
DECL E6POS POPE3={X 363.888,Y 19.3187675,Z 1.50000,A 0.0,B 0.0,C 20.0000}
DECL FDAT FPE3={TOOL_NO 2,BASE_NO 2,IPO_FRAME #BASE,POINT2[] " ",TQ_STATE FALSE}
DECL LDAT LPM3={VEL 0.0230000,ACC 100.000,APO_DIST 5.00000,APO_FAC 50.0000,AXIS_VEL 100.000,AXIS_ACC 100.000,ORI_TYP #VAR,CIRC_TYP #BASE,JERK_FAC 50.0000,GEAR_JERK 50.0000,EXAX_IGN 0}
DECL E6POS POS6={X 32.1370,Y -0.736000,Z -150.000,A 0.0,B 0.0,C 0.0}
DECL FDAT FS6={TOOL_NO 2,BASE_NO 2,IPO_FRAME #BASE,POINT2[] " ",TQ_STATE FALSE}
DECL LDAT LL6={VEL 0.500000,ACC 100.000,APO_DIST 0.0,APO_FAC 50.0000,AXIS_VEL 100.000,AXIS_ACC 100.000,ORI_TYP #VAR,CIRC_TYP #BASE,JERK_FAC 50.0000,GEAR_JERK 50.0000,EXAX_IGN 0}
DECL E6POS POS7={X 32.1370,Y -0.736000,Z 0.0,A 0.0,B 0.0,C 0.0}
DECL FDAT FS7={TOOL_NO 2,BASE_NO 2,IPO_FRAME #BASE,POINT2[] " ",TQ_STATE FALSE}
DECL LDAT LL7={VEL 0.500000,ACC 100.000,APO_DIST 0.0,APO_FAC 50.0000,AXIS_VEL 100.000,AXIS_ACC 100.000,ORI_TYP #VAR,CIRC_TYP #BASE,JERK_FAC 50.0000,GEAR_JERK 50.0000,EXAX_IGN 0}
DECL E6POS POS8={X 32.1600,Y 18.4470,Z 0.0,A 0.0,B 0.0,C 0.0}
DECL FDAT FS8={TOOL_NO 2,BASE_NO 2,IPO_FRAME #BASE,POINT2[] " ",TQ_STATE FALSE}
DECL LDAT LL8={VEL 0.01000000,ACC 100.000,APO_DIST 0.0,APO_FAC 50.0000,AXIS_VEL 100.000,AXIS_ACC 100.000,ORI_TYP #VAR,CIRC_TYP #BASE,JERK_FAC 50.0000,GEAR_JERK 50.0000,EXAX_IGN 0}
DECL E6POS POS9={X 32.1485,Y 8.85550117,Z -150.000,A 0.0,B 0.0,C 0.0}
DECL FDAT FS9={TOOL_NO 2,BASE_NO 2,IPO_FRAME #BASE,POINT2[] " ",TQ_STATE FALSE}
DECL LDAT LL9={VEL 0.500000,ACC 100.000,APO_DIST 0.0,APO_FAC 50.0000,AXIS_VEL 100.000,AXIS_ACC 100.000,ORI_TYP #VAR,CIRC_TYP #BASE,JERK_FAC 50.0000,GEAR_JERK 50.0000,EXAX_IGN 0}
DECL E6POS POPM4={X 23.1220,Y 21.6800,Z 1.50000,A 0.0,B 0.0,C 0.0}
DECL E6POS POPE4={X 18.7403107,Y 31.1279984,Z 1.50000,A 0.0,B -20.0000,C 0.0}
DECL FDAT FPE4={TOOL_NO 2,BASE_NO 2,IPO_FRAME #BASE,POINT2[] " ",TQ_STATE FALSE}
DECL LDAT LPM4={VEL 0.0120000,ACC 100.000,APO_DIST 5.00000,APO_FAC 50.0000,AXIS_VEL 100.000,AXIS_ACC 100.000,ORI_TYP #VAR,CIRC_TYP #BASE,JERK_FAC 50.0000,GEAR_JERK 50.0000,EXAX_IGN 0}
DECL E6POS POPM5={X 22.5580,Y 657.793,Z 1.50000,A 0.0,B 0.0,C 0.0}
DECL E6POS POPE5={X 30.8369904,Y 660.939636,Z 0.500000,A 0.0,B 0.0,C -20.0000}
DECL FDAT FPE5={TOOL_NO 2,BASE_NO 2,IPO_FRAME #BASE,POINT2[] " ",TQ_STATE FALSE}
DECL LDAT LPM5={VEL 0.0120000,ACC 100.000,APO_DIST 5.00000,APO_FAC 50.0000,AXIS_VEL 100.000,AXIS_ACC 100.000,ORI_TYP #VAR,CIRC_TYP #BASE,JERK_FAC 50.0000,GEAR_JERK 50.0000,EXAX_IGN 0}
DECL E6POS POPM7={X 370.952026,Y 658.128,Z 2.50000,A 0.0,B 0.0,C 0.0}
DECL E6POS POPE7={X 375.437683,Y 649.261047,Z 2.50000,A 0.0,B 20.0000,C 0.0}
DECL FDAT FPE7={TOOL_NO 2,BASE_NO 2,IPO_FRAME #BASE,POINT2[] " ",TQ_STATE FALSE}
DECL LDAT LPM7={VEL 0.0120000,ACC 100.000,APO_DIST 5.00000,APO_FAC 50.0000,AXIS_VEL 100.000,AXIS_ACC 100.000,ORI_TYP #VAR,CIRC_TYP #BASE,JERK_FAC 50.0000,GEAR_JERK 50.0000,EXAX_IGN 0}
DECL E6POS POS10={X 31.6630,Y 678.803,Z -150.000,A 0.0,B 0.0,C 0.0}
DECL FDAT FS10={TOOL_NO 2,BASE_NO 2,IPO_FRAME #BASE,POINT2[] " ",TQ_STATE FALSE}
DECL LDAT LL10={VEL 0.500000,ACC 100.000,APO_DIST 0.0,APO_FAC 50.0000,AXIS_VEL 100.000,AXIS_ACC 100.000,ORI_TYP #VAR,CIRC_TYP #BASE,JERK_FAC 50.0000,GEAR_JERK 50.0000,EXAX_IGN 0}
DECL E6POS POS11={X 31.6630,Y 678.803,Z 0.0,A 0.0,B 0.0,C 0.0}
DECL FDAT FS11={TOOL_NO 2,BASE_NO 2,IPO_FRAME #BASE,POINT2[] " ",TQ_STATE FALSE}
DECL LDAT LL11={VEL 0.500000,ACC 100.000,APO_DIST 0.0,APO_FAC 50.0000,AXIS_VEL 100.000,AXIS_ACC 100.000,ORI_TYP #VAR,CIRC_TYP #BASE,JERK_FAC 50.0000,GEAR_JERK 50.0000,EXAX_IGN 0}
DECL E6POS POS12={X 31.3610,Y 659.596,Z 0.0,A 0.0,B 0.0,C 0.0}
DECL FDAT FS12={TOOL_NO 2,BASE_NO 2,IPO_FRAME #BASE,POINT2[] " ",TQ_STATE FALSE}
DECL LDAT LL12={VEL 0.01000000,ACC 100.000,APO_DIST 0.0,APO_FAC 50.0000,AXIS_VEL 100.000,AXIS_ACC 100.000,ORI_TYP #VAR,CIRC_TYP #BASE,JERK_FAC 50.0000,GEAR_JERK 50.0000,EXAX_IGN 0}
DECL E6POS POS13={X 31.5120010,Y 669.199463,Z -150.000,A 0.0,B 0.0,C 0.0}
DECL FDAT FS13={TOOL_NO 2,BASE_NO 2,IPO_FRAME #BASE,POINT2[] " ",TQ_STATE FALSE}
DECL LDAT LL13={VEL 0.500000,ACC 100.000,APO_DIST 0.0,APO_FAC 50.0000,AXIS_VEL 100.000,AXIS_ACC 100.000,ORI_TYP #VAR,CIRC_TYP #BASE,JERK_FAC 50.0000,GEAR_JERK 50.0000,EXAX_IGN 0}
DECL E6POS POS14={X 361.885,Y 679.437,Z -150.000,A 0.0,B 0.0,C 0.0}
DECL FDAT FS14={TOOL_NO 2,BASE_NO 2,IPO_FRAME #BASE,POINT2[] " ",TQ_STATE FALSE}
DECL LDAT LL14={VEL 0.500000,ACC 100.000,APO_DIST 0.0,APO_FAC 50.0000,AXIS_VEL 100.000,AXIS_ACC 100.000,ORI_TYP #VAR,CIRC_TYP #BASE,JERK_FAC 50.0000,GEAR_JERK 50.0000,EXAX_IGN 0}
DECL E6POS POS15={X 361.885,Y 679.437,Z 1.00000,A 0.0,B 0.0,C 0.0}
DECL FDAT FS15={TOOL_NO 2,BASE_NO 2,IPO_FRAME #BASE,POINT2[] " ",TQ_STATE FALSE}
DECL LDAT LL15={VEL 0.500000,ACC 100.000,APO_DIST 0.0,APO_FAC 50.0000,AXIS_VEL 100.000,AXIS_ACC 100.000,ORI_TYP #VAR,CIRC_TYP #BASE,JERK_FAC 50.0000,GEAR_JERK 50.0000,EXAX_IGN 0}
DECL E6POS POS16={X 361.560,Y 660.457,Z 1.00000,A 0.0,B 0.0,C 0.0}
DECL FDAT FS16={TOOL_NO 2,BASE_NO 2,IPO_FRAME #BASE,POINT2[] " ",TQ_STATE FALSE}
DECL LDAT LL16={VEL 0.01000000,ACC 100.000,APO_DIST 0.0,APO_FAC 50.0000,AXIS_VEL 100.000,AXIS_ACC 100.000,ORI_TYP #VAR,CIRC_TYP #BASE,JERK_FAC 50.0000,GEAR_JERK 50.0000,EXAX_IGN 0}
DECL E6POS POS17={X 361.722504,Y 669.947,Z -150.000,A 0.0,B 0.0,C 0.0}
DECL FDAT FS17={TOOL_NO 2,BASE_NO 2,IPO_FRAME #BASE,POINT2[] " ",TQ_STATE FALSE}
DECL LDAT LL17={VEL 0.500000,ACC 100.000,APO_DIST 0.0,APO_FAC 50.0000,AXIS_VEL 100.000,AXIS_ACC 100.000,ORI_TYP #VAR,CIRC_TYP #BASE,JERK_FAC 50.0000,GEAR_JERK 50.0000,EXAX_IGN 0}
DECL PDAT PPDAT3={VEL 100.000,ACC 20.0000,APO_DIST 100.000,APO_MODE #CDIS,GEAR_JERK 50.0000,EXAX_IGN 0}
DECL FDAT FL0_S2={TOOL_NO 2,BASE_NO 2,IPO_FRAME #BASE,POINT2[] " ",TQ_STATE FALSE}
DECL E6POS POL0_S2={X 375.372040,Y 587.535706,Z 2.50000,A 0.0,B 20.0000,C 0.0}
DECL FDAT FL0={TOOL_NO 2,BASE_NO 11,IPO_FRAME #BASE,POINT2[] " ",TQ_STATE FALSE}
DECL E6POS POL0_s4={X 375.681305,Y 31.1079712,Z 2.50000,A 0.0,B 20.0000,C 0.0}
DECL FDAT FL0_s4={TOOL_NO 2,BASE_NO 2,IPO_FRAME #BASE,POINT2[] " ",TQ_STATE FALSE}
DECL E6POS POC45_S5={X 404.000,Y 36.0000,Z -1.00000,A 0.0,B 20.0000,C 0.0}
DECL FDAT FC45_S5={TOOL_NO 2,BASE_NO 11,IPO_FRAME #BASE,POINT2[] " ",TQ_STATE FALSE}
DECL E6POS POL0_S1={X 375.946960,Y 92.9332886,Z 2.50000,A 0.0,B 20.0000,C 0.0}
DECL FDAT FL0_S1={TOOL_NO 2,BASE_NO 2,IPO_FRAME #BASE,POINT2[] " ",TQ_STATE FALSE}
DECL E6POS POC45_S1={X 375.881317,Y 31.1079712,Z 1.50000,A 0.0,B 20.0000,C 0.0}
DECL FDAT FC45_S1={TOOL_NO 2,BASE_NO 2,IPO_FRAME #BASE,POINT2[] " ",TQ_STATE FALSE}
DECL LDAT LL0_L1={VEL 0.300000,ACC 100.000,APO_DIST 5.00000,APO_FAC 50.0000,AXIS_VEL 100.000,AXIS_ACC 100.000,ORI_TYP #VAR,CIRC_TYP #BASE,JERK_FAC 50.0000,GEAR_JERK 50.0000,EXAX_IGN 0}
DECL LDAT LC45_L1={VEL 0.300000,ACC 100.000,APO_DIST 5.00000,APO_FAC 50.0000,AXIS_VEL 100.000,AXIS_ACC 100.000,ORI_TYP #VAR,CIRC_TYP #BASE,JERK_FAC 50.0000,GEAR_JERK 50.0000,EXAX_IGN 0}
DECL E6POS POL90_S1={X 330.624,Y 19.5486126,Z 1.50000,A 0.0,B 0.0,C 20.0000}
DECL FDAT FL90_S1={TOOL_NO 2,BASE_NO 2,IPO_FRAME #BASE,POINT2[] " ",TQ_STATE FALSE}
DECL LDAT LL90_L1={VEL 0.0250000,ACC 100.000,APO_DIST 5.00000,APO_FAC 50.0000,AXIS_VEL 100.000,AXIS_ACC 100.000,ORI_TYP #VAR,CIRC_TYP #BASE,JERK_FAC 50.0000,GEAR_JERK 50.0000,EXAX_IGN 0}
DECL E6POS POL90_S2={X 197.568,Y 19.2680,Z 1.50000,A 0.0,B 0.0,C 20.0000}
DECL FDAT FL90_S2={TOOL_NO 2,BASE_NO 2,IPO_FRAME #BASE,POINT2[] " ",TQ_STATE FALSE}
DECL LDAT LL90_L2={VEL 0.0250000,ACC 100.000,APO_DIST 5.00000,APO_FAC 50.0000,AXIS_VEL 100.000,AXIS_ACC 100.000,ORI_TYP #VAR,CIRC_TYP #BASE,JERK_FAC 50.0000,GEAR_JERK 50.0000,EXAX_IGN 0}
DECL E6POS POL90_S3={X 64.5119934,Y 18.9873867,Z 1.50000,A 0.0,B 0.0,C 20.0000}
DECL FDAT FL90_S3={TOOL_NO 2,BASE_NO 2,IPO_FRAME #BASE,POINT2[] " ",TQ_STATE FALSE}
DECL LDAT LL90_L3={VEL 0.0250000,ACC 100.000,APO_DIST 5.00000,APO_FAC 50.0000,AXIS_VEL 100.000,AXIS_ACC 100.000,ORI_TYP #VAR,CIRC_TYP #BASE,JERK_FAC 50.0000,GEAR_JERK 50.0000,EXAX_IGN 0}
DECL E6POS POC135_S1={X 31.2479858,Y 19.1172333,Z 1.50000,A 0.0,B 0.0,C 20.0000}
DECL FDAT FC135_S1={TOOL_NO 2,BASE_NO 2,IPO_FRAME #BASE,POINT2[] " ",TQ_STATE FALSE}
DECL LDAT LC135_L1={VEL 0.200000,ACC 50.0000,APO_DIST 5.00000,APO_FAC 50.0000,AXIS_VEL 100.000,AXIS_ACC 100.000,ORI_TYP #VAR,CIRC_TYP #BASE,JERK_FAC 50.0000,GEAR_JERK 50.0000,EXAX_IGN 0}
DECL E6POS POL180_S1={X 18.5007477,Y 93.1777,Z 1.50000,A 0.0,B -20.0000,C 0.0}
DECL FDAT FL180_S1={TOOL_NO 2,BASE_NO 2,IPO_FRAME #BASE,POINT2[] " ",TQ_STATE FALSE}
DECL LDAT LL180_L1={VEL 0.0250000,ACC 100.000,APO_DIST 5.00000,APO_FAC 50.0000,AXIS_VEL 100.000,AXIS_ACC 100.000,ORI_TYP #VAR,CIRC_TYP #BASE,JERK_FAC 50.0000,GEAR_JERK 50.0000,EXAX_IGN 0}
DECL E6POS POL180_S2={X 18.7425,Y 340.176514,Z 1.50000,A 0.0,B -20.0000,C 0.0}
DECL FDAT FL180_S2={TOOL_NO 2,BASE_NO 2,IPO_FRAME #BASE,POINT2[] " ",TQ_STATE FALSE}
DECL LDAT LL180_L2={VEL 0.0300000,ACC 100.000,APO_DIST 5.00000,APO_FAC 50.0000,AXIS_VEL 100.000,AXIS_ACC 100.000,ORI_TYP #VAR,CIRC_TYP #BASE,JERK_FAC 50.0000,GEAR_JERK 50.0000,EXAX_IGN 0}
DECL E6POS POL180_S3={X 18.3644695,Y 618.050110,Z 1.50000,A 0.0,B -20.0000,C 0.0}
DECL FDAT FL180_S3={TOOL_NO 2,BASE_NO 2,IPO_FRAME #BASE,POINT2[] " ",TQ_STATE FALSE}
DECL LDAT LL180_L3={VEL 0.0300000,ACC 100.000,APO_DIST 5.00000,APO_FAC 50.0000,AXIS_VEL 100.000,AXIS_ACC 100.000,ORI_TYP #VAR,CIRC_TYP #BASE,JERK_FAC 50.0000,GEAR_JERK 50.0000,EXAX_IGN 0}
DECL E6POS POC225_S1={X 18.6446877,Y 648.925,Z 1.50000,A 0.0,B -20.0000,C 0.0}
DECL FDAT FC225_S1={TOOL_NO 2,BASE_NO 2,IPO_FRAME #BASE,POINT2[] " ",TQ_STATE FALSE}
DECL LDAT LC225_L1={VEL 0.200000,ACC 50.0000,APO_DIST 5.00000,APO_FAC 50.0000,AXIS_VEL 100.000,AXIS_ACC 100.000,ORI_TYP #VAR,CIRC_TYP #BASE,JERK_FAC 50.0000,GEAR_JERK 50.0000,EXAX_IGN 0}
DECL E6POS POL270_S1={X 64.1063919,Y 660.880310,Z 0.500000,A 0.0,B 0.0,C -20.0000}
DECL FDAT FL270_S1={TOOL_NO 2,BASE_NO 2,IPO_FRAME #BASE,POINT2[] " ",TQ_STATE FALSE}
DECL LDAT Ll270_L1={VEL 0.0250000,ACC 100.000,APO_DIST 5.00000,APO_FAC 50.0000,AXIS_VEL 100.000,AXIS_ACC 100.000,ORI_TYP #VAR,CIRC_TYP #BASE,JERK_FAC 50.0000,GEAR_JERK 50.0000,EXAX_IGN 0}
DECL E6POS POL270_S2={X 197.184,Y 660.843,Z 1.50000,A 0.0,B 0.0,C -20.0000}
DECL FDAT FL270_S2={TOOL_NO 2,BASE_NO 2,IPO_FRAME #BASE,POINT2[] " ",TQ_STATE FALSE}
DECL LDAT LL270_L2={VEL 0.0300000,ACC 100.000,APO_DIST 5.00000,APO_FAC 50.0000,AXIS_VEL 100.000,AXIS_ACC 100.000,ORI_TYP #VAR,CIRC_TYP #BASE,JERK_FAC 50.0000,GEAR_JERK 50.0000,EXAX_IGN 0}
DECL E6POS POL270_S3={X 346.896301,Y 660.926,Z 1.50000,A 0.0,B 0.0,C -20.0000}
DECL FDAT FL270_S3={TOOL_NO 2,BASE_NO 2,IPO_FRAME #BASE,POINT2[] " ",TQ_STATE FALSE}
DECL LDAT LL270_L3={VEL 0.0300000,ACC 100.000,APO_DIST 5.00000,APO_FAC 50.0000,AXIS_VEL 100.000,AXIS_ACC 100.000,ORI_TYP #VAR,CIRC_TYP #BASE,JERK_FAC 50.0000,GEAR_JERK 50.0000,EXAX_IGN 0}
DECL E6POS POC315_S1={X 363.531,Y 660.846375,Z 0.0,A 0.0,B 0.0,C -20.0000}
DECL FDAT FC315_S1={TOOL_NO 2,BASE_NO 2,IPO_FRAME #BASE,POINT2[] " ",TQ_STATE FALSE}
DECL LDAT LC315_L1={VEL 0.200000,ACC 50.0000,APO_DIST 5.00000,APO_FAC 50.0000,AXIS_VEL 100.000,AXIS_ACC 100.000,ORI_TYP #VAR,CIRC_TYP #BASE,JERK_FAC 50.0000,GEAR_JERK 50.0000,EXAX_IGN 0}
DECL LDAT LL0_L2={VEL 0.0300000,ACC 100.000,APO_DIST 5.00000,APO_FAC 50.0000,AXIS_VEL 100.000,AXIS_ACC 100.000,ORI_TYP #VAR,CIRC_TYP #BASE,JERK_FAC 50.0000,GEAR_JERK 50.0000,EXAX_IGN 0}
DECL E6POS POL0_S3={X 375.409515,Y 340.234497,Z 2.50000,A 0.0,B 20.0000,C 0.0}
DECL FDAT FL0_S3={TOOL_NO 2,BASE_NO 2,IPO_FRAME #BASE,POINT2[] " ",TQ_STATE FALSE}
DECL LDAT LL0_L3={VEL 0.0300000,ACC 100.000,APO_DIST 5.00000,APO_FAC 50.0000,AXIS_VEL 100.000,AXIS_ACC 100.000,ORI_TYP #VAR,CIRC_TYP #BASE,JERK_FAC 50.0000,GEAR_JERK 50.0000,EXAX_IGN 0}
DECL LDAT LL0_L4={VEL 0.0400000,ACC 100.000,APO_DIST 5.00000,APO_FAC 50.0000,AXIS_VEL 100.000,AXIS_ACC 100.000,ORI_TYP #VAR,CIRC_TYP #BASE,JERK_FAC 50.0000,GEAR_JERK 50.0000,EXAX_IGN 0}
DECL E6POS XP2={X 293.122131,Y 89.9176636,Z -80.0293961,A 0.0,B 0.0,C 0.0,S 2,T 10,E1 0.0,E2 0.0,E3 0.0,E4 0.0,E5 0.0,E6 0.0}
DECL FDAT Fp2={TOOL_NO 2,BASE_NO 2,IPO_FRAME #BASE,POINT2[] " "}
DECL LDAT LCPDAT1={VEL 0.500000,ACC 50.0000,APO_DIST 100.000,APO_FAC 50.0000,AXIS_VEL 100.000,AXIS_ACC 100.000,ORI_TYP #VAR,CIRC_TYP #BASE,JERK_FAC 50.0000,GEAR_JERK 50.0000,EXAX_IGN 0,CB {AUX_PT {ORI #CONSIDER,E1 #CONSIDER,E2 #CONSIDER,E3 #CONSIDER,E4 #CONSIDER,E5 #CONSIDER,E6 #CONSIDER},TARGET_PT {ORI #INTERPOLATE,E1 #INTERPOLATE,E2 #INTERPOLATE,E3 #INTERPOLATE,E4 #INTERPOLATE,E5 #INTERPOLATE,E6 #INTERPOLATE}}}
DECL E6POS XP3={X -42.3839874,Y 91.8151550,Z -80.0254822,A 0.0,B 0.0,C 0.0,S 2,T 10,E1 0.0,E2 0.0,E3 0.0,E4 0.0,E5 0.0,E6 0.0}
DECL FDAT Fp3={TOOL_NO 2,BASE_NO 2,IPO_FRAME #BASE,POINT2[] " "}
DECL LDAT LCPDAT2={VEL 0.500000,ACC 50.0000,APO_DIST 100.000,APO_FAC 50.0000,AXIS_VEL 100.000,AXIS_ACC 100.000,ORI_TYP #VAR,CIRC_TYP #BASE,JERK_FAC 50.0000,GEAR_JERK 50.0000,EXAX_IGN 0,CB {AUX_PT {ORI #CONSIDER,E1 #CONSIDER,E2 #CONSIDER,E3 #CONSIDER,E4 #CONSIDER,E5 #CONSIDER,E6 #CONSIDER},TARGET_PT {ORI #INTERPOLATE,E1 #INTERPOLATE,E2 #INTERPOLATE,E3 #INTERPOLATE,E4 #INTERPOLATE,E5 #INTERPOLATE,E6 #INTERPOLATE}}}
DECL E6POS XP4={X -39.7999954,Y 716.082336,Z -80.0293350,A 0.0,B 0.0,C 0.0,S 2,T 43,E1 0.0,E2 0.0,E3 0.0,E4 0.0,E5 0.0,E6 0.0}
DECL FDAT Fp4={TOOL_NO 2,BASE_NO 2,IPO_FRAME #BASE,POINT2[] " "}
DECL LDAT LCPDAT3={VEL 0.500000,ACC 50.0000,APO_DIST 100.000,APO_FAC 50.0000,AXIS_VEL 100.000,AXIS_ACC 100.000,ORI_TYP #VAR,CIRC_TYP #BASE,JERK_FAC 50.0000,GEAR_JERK 50.0000,EXAX_IGN 0,CB {AUX_PT {ORI #CONSIDER,E1 #CONSIDER,E2 #CONSIDER,E3 #CONSIDER,E4 #CONSIDER,E5 #CONSIDER,E6 #CONSIDER},TARGET_PT {ORI #INTERPOLATE,E1 #INTERPOLATE,E2 #INTERPOLATE,E3 #INTERPOLATE,E4 #INTERPOLATE,E5 #INTERPOLATE,E6 #INTERPOLATE}}}
DECL E6POS XP5={X 294.984924,Y 714.198059,Z -80.0293350,A 0.0,B 0.0,C 0.0,S 2,T 43,E1 0.0,E2 0.0,E3 0.0,E4 0.0,E5 0.0,E6 0.0}
DECL FDAT Fp5={TOOL_NO 2,BASE_NO 2,IPO_FRAME #BASE,POINT2[] " "}
DECL LDAT LCPDAT4={VEL 0.500000,ACC 50.0000,APO_DIST 100.000,APO_FAC 50.0000,AXIS_VEL 100.000,AXIS_ACC 100.000,ORI_TYP #VAR,CIRC_TYP #BASE,JERK_FAC 50.0000,GEAR_JERK 50.0000,EXAX_IGN 0,CB {AUX_PT {ORI #CONSIDER,E1 #CONSIDER,E2 #CONSIDER,E3 #CONSIDER,E4 #CONSIDER,E5 #CONSIDER,E6 #CONSIDER},TARGET_PT {ORI #INTERPOLATE,E1 #INTERPOLATE,E2 #INTERPOLATE,E3 #INTERPOLATE,E4 #INTERPOLATE,E5 #INTERPOLATE,E6 #INTERPOLATE}}}
DECL PDAT PPDAT4={VEL 10.0000,ACC 20.0000,APO_DIST 100.000,APO_MODE #CDIS,GEAR_JERK 50.0000,EXAX_IGN 0}
DECL MODULEPARAM_T LAST_TP_PARAMS={PARAMS[] "LASER_FUNCTION.LSPOW=100; LASER_FUNCTION.LSSEC=0; SURROUND_LIN.MOVE_NAME=L0_S4; SURROUND_LIN.VEL=0.04; SURROUND_LIN.LIN_POSITION=100; SURROUND_LIN.AREA_LIN_LIST=L0; SURROUND_LIN.MOVE_LDAT=L0_L4; SURROUND_LIN.OFFSET_NO=4; SURROUND_LIN.WORK_AREA=2; SURROUND_LIN.AREA_CIR_LIST=C45; SURROUND_CIR.CIR_MID_NAME=PM7; SURROUND_CIR.CIR_END_NAME=PE7; SURROUND_CIR.VEL=0.012; SURROUND_CIR.AREA_CIR_LIST=C315; SURROUND_CIR.WORK_AREA=2; SHORT_CRAFT.MOVE_NAME=S17; SHORT_CRAFT.VEL=0.5; SHORT_CRAFT.AREA_LIN_LIST=N315; SHORT_CRAFT.SHORT_POS=4; SHORT_CRAFT.LIN_POSITION=50; SHORT_CRAFT.MOVE_LDAT=L17; SHORT_CRAFT.WORK_AREA=2; Kuka.PointName=p5; Kuka.FrameData.base_no=2; Kuka.FrameData.tool_no=2; Kuka.FrameData.ipo_frame=#BASE; Kuka.FrameData.point2=; Kuka.isglobalpoint=False; Kuka.MoveDataName=CPDAT4; Kuka.MovementData.cb={AUX_PT {ORI #CONSIDER,E1 #CONSIDER,E2 #CONSIDER,E3 #CONSIDER,E4 #CONSIDER,E5 #CONSIDER,E6 #CONSIDER},TARGET_PT {ORI #INTERPOLATE,E1 #INTERPOLATE,E2 #INTERPOLATE,E3 #INTERPOLATE,E4 #INTERPOLATE,E5 #INTERPOLATE,E6 #INTERPOLATE}}; Kuka.MovementData.apo_fac=50; Kuka.MovementData.apo_dist=100; Kuka.MovementData.axis_acc=100; Kuka.MovementData.axis_vel=100; Kuka.MovementData.circ_typ=#BASE; Kuka.MovementData.jerk_fac=50; Kuka.MovementData.ori_typ=#VAR; Kuka.MovementData.vel=10; Kuka.MovementData.acc=20; Kuka.MovementData.exax_ign=0; Kuka.VelocityPath=0.5; Kuka.BlendingEnabled=False; Kuka.APXEnabled=False; Kuka.CurrentCDSetIndex=0; Kuka.MoveDataPtpName=PDAT4                    "}
DECL LDAT LL1={VEL 0.200000,ACC 50.0000,APO_DIST 5.00000,APO_FAC 50.0000,AXIS_VEL 100.000,AXIS_ACC 100.000,ORI_TYP #VAR,CIRC_TYP #BASE,JERK_FAC 50.0000,GEAR_JERK 50.0000,EXAX_IGN 0}
DECL LDAT LL18={VEL 0.200000,ACC 50.0000,APO_DIST 5.00000,APO_FAC 50.0000,AXIS_VEL 100.000,AXIS_ACC 100.000,ORI_TYP #VAR,CIRC_TYP #BASE,JERK_FAC 50.0000,GEAR_JERK 50.0000,EXAX_IGN 0}
DECL FDAT FS1={TOOL_NO 2,BASE_NO 2,IPO_FRAME #BASE,POINT2[] " ",TQ_STATE FALSE}
DECL LDAT LL19={VEL 0.200000,ACC 50.0000,APO_DIST 5.00000,APO_FAC 50.0000,AXIS_VEL 100.000,AXIS_ACC 100.000,ORI_TYP #VAR,CIRC_TYP #BASE,JERK_FAC 50.0000,GEAR_JERK 50.0000,EXAX_IGN 0}
DECL E6POS POS1={X 375.158691,Y 92.2952271,Z 1.00000,A 0.0,B -20.0000,C 0.0}
DECL MODULEPARAM_T LAST_TP_PARAMS2={PARAMS[] "Kuka.MovementDataPdat.apo_mode=#CDIS; Kuka.MovementDataPdat.apo_dist=100; Kuka.VelocityPtp=10                    "}
ENDDAT
